(*
SPDX-FileCopyrightText: © 2026 Oleksandr Tiutyk <trofimich@gmail.com>
SPDX-License-Identifier: MIT
License: https://opensource.org/license/mit
*)

FUNCTION_BLOCK VARIABLE_DESCRIPTOR
VAR_OUTPUT	
	Name : STRING;
	TypeClass : TOF_Core.GENERIC_TYPE_CLASS;
	Address : PVOID;
	Size : ULINT;
END_VAR

METHOD Initialize
VAR_INPUT
	variableName : STRING;
	plcVariable : ANY;
	plcVariableIsObject : BOOL := FALSE;
END_VAR
VAR
	workflowVariableNameEmptyException : TOF_Core.ArgumentOutOfRangeException;
END_VAR
IF variableName = '' THEN
	workflowVariableNameEmptyException.Throw(CurrentNamespace.Name, 'VARIABLE_DESCRIPTOR', __POUNAME(), __POSITION(), 'variableName', variableName);
END_IF

Name := variableName;
TypeClass := TOF_Core.GenericTypeClassConvertor.GetGenericTypeClassBySystemAnyType(plcVariable, plcVariableIsObject);
Address := plcVariable.pValue;
Size := TO_ULINT(plcVariable.diSize);
END_METHOD

END_FUNCTION_BLOCK

(* stored: Version 1.1.0.1
   POU VARIABLE_DESCRIPTOR: Id {21b7987f-8a83-4a82-8f93-778006b20007}, SpecialFunc None
   Method Initialize: Id {72a9a034-b16f-4dea-be41-e77dfe5fa87a} *)
